{attribute addProperty BoxType "EL2212-0000-0018"}
{attribute addProperty Id "OutputBIT10.1252TristateBIT10.1253ResetBIT10.1258"}
{attribute addProperty CRC "1242702358"}
{attribute addProperty SizeInBites "16"}
{attribute addProperty SizeInBytes "2"}
TYPE Control_4A122216 :
STRUCT
	{attribute 'hide'}
	reserve_1 : BIT;
	{attribute addProperty Name "Output"}
	Output : BIT;
	{attribute addProperty Name "Tristate"}
	Tristate : BIT;
	{attribute 'hide'}
	reserve_2_BIT_0 : BIT;
	{attribute 'hide'}
	reserve_2_BIT_1 : BIT;
	{attribute 'hide'}
	reserve_2_BIT_2 : BIT;
	{attribute 'hide'}
	reserve_2_BIT_3 : BIT;
	{attribute addProperty Name "Reset"}
	Reset : BIT;
	{attribute 'hide'}
	reserve_3 : BYTE;
END_STRUCT
END_TYPE

(* stored: Version 1.2.0.0, ProductVersion 3.1.4024.9
   DUT Control_4A122216: Id {079a74b3-327b-44ee-84a5-adb1c2d299a2} *)
